PROGRAM MAIN
VAR
	a:INT;
	b:INT;
	c:INT;
	add1:FB_ADD;
END_VAR

add1(in1:=a ,in2:=b , out =>c );

END_PROGRAM

(* stored: Version 1.1.0.1, ProductVersion 3.1.4024.11
   POU MAIN: Id {c7c736b2-d542-4c88-91fe-68de5eef900f}, SpecialFunc None *)
